# EPICS substitutions: example/exampleApp/Db/posCompEx.substitutions
file positioncompare.template
{
pattern { P, PORT, PLC }
		{ P, pmac_S0, 15 }
}
